TYPE ST_DigitalOutput_IO :
STRUCT
    outSignal : BOOL;
END_STRUCT
END_TYPE

(* stored: Version 1.1.0.1, ProductVersion 3.1.4026.12
   DUT ST_DigitalOutput_IO: Id {b0100002-0003-0000-0000-000000000001} *)
